# B&R Automation Studio project Lab1FuncBlocks
Automation Studio 4.5.2.102

## Configuration Config1

### Task classes (Cpu.sw)
```
Cyclic#4:
  Program <- Program.prg
Libraries: MotorCntrl
```

### Hardware
```
4PP065_0571_P74 : 4PP065.0571-P74 v1.1.2.0
  Simulation = 1
```

## Logical view

### Library Logical/Libraries/MotorCntrl (ANSIC)

#### MotorCntrl.fun - Exported functions and function blocks
```iecst
{REDUND_ERROR} {REDUND_UNREPLICABLE} FUNCTION_BLOCK FB_Motor (*Motor Model*) (*$GROUP=User,$CAT=User,$GROUPICON=User.png,$CATICON=User.png*)
	VAR_INPUT
		u : {REDUND_UNREPLICABLE} REAL; (*input voltage*)
	END_VAR
	VAR_OUTPUT
		w : {REDUND_UNREPLICABLE} REAL; (*rotation speed*)
		phi : {REDUND_UNREPLICABLE} REAL; (*position*)
	END_VAR
	VAR
		integrator : {REDUND_UNREPLICABLE} FB_Integrator; (*integrator*)
		Tm : {REDUND_UNREPLICABLE} REAL; (*Tm*)
		Ke : {REDUND_UNREPLICABLE} REAL; (*Ke*)
		dt : {REDUND_UNREPLICABLE} REAL; (*calc step*)
	END_VAR
END_FUNCTION_BLOCK

{REDUND_ERROR} {REDUND_UNREPLICABLE} FUNCTION_BLOCK FB_Integrator (*Integrator*) (*$GROUP=User,$CAT=User,$GROUPICON=User.png,$CATICON=User.png*)
	VAR_INPUT
		in : {REDUND_UNREPLICABLE} REAL; (*inp_integrator*)
	END_VAR
	VAR_OUTPUT
		out : {REDUND_UNREPLICABLE} REAL; (*out_integrator*)
	END_VAR
	VAR
		dt : {REDUND_UNREPLICABLE} REAL; (*calc_step*)
	END_VAR
END_FUNCTION_BLOCK

{REDUND_ERROR} FUNCTION_BLOCK FB_Regulator (*PI regulator*) (*$GROUP=User,$CAT=User,$GROUPICON=User.png,$CATICON=User.png*)
	VAR_INPUT
		e : {REDUND_UNREPLICABLE} REAL; (*Disagreement*)
	END_VAR
	VAR_OUTPUT
		u : {REDUND_UNREPLICABLE} REAL; (*voltage *)
	END_VAR
	VAR
		K_p : {REDUND_UNREPLICABLE} REAL; (*K_p*)
		K_i : {REDUND_UNREPLICABLE} REAL; (*K_i*)
		integrator : {REDUND_UNREPLICABLE} FB_Integrator; (*integrator*)
		iyOld : {REDUND_UNREPLICABLE} REAL; (*storing the value*)
		max_abs_value : {REDUND_UNREPLICABLE} REAL; (*edge of restriction block*)
		dt : {REDUND_UNREPLICABLE} REAL; (*calc_step*)
	END_VAR
END_FUNCTION_BLOCK
```

#### FB_Motor.c
```c
#include <bur/plctypes.h>
#ifdef __cplusplus
	extern "C"
	{
#endif
	#include "MotorCntrl.h"
#ifdef __cplusplus
	};
#endif
/* Motor Model */
void FB_Motor(struct FB_Motor* inst)
{
	inst->integrator.in = (inst->u / inst->Ke - inst->w) * inst->dt / inst->Tm;
	FB_Integrator(&(inst->integrator));
	inst->w = inst->integrator.out;
	inst->integrator.in = inst->w * inst->dt;
	FB_Integrator(&(inst->integrator));
	inst->phi = inst->integrator.out;
}
```

#### FB_Integrator.c
```c
#include <bur/plctypes.h>
#ifdef __cplusplus
	extern "C"
	{
#endif
	#include "MotorCntrl.h"
#ifdef __cplusplus
	};
#endif
/* Integrator */
void FB_Integrator(struct FB_Integrator* inst)
{
	inst->out +=  inst->in;
}
```

#### FB_Regulator.c
```c
#include <bur/plctypes.h>
#ifdef __cplusplus
	extern "C"
	{
#endif
	#include "MotorCntrl.h"
#ifdef __cplusplus
	};
#endif

void FB_Regulator(struct FB_Regulator* inst)
{

	REAL in_BON=0; REAL sum_after = 0;
	inst->integrator.in=inst->e * inst->K_i * inst->dt + inst->iyOld;
	FB_Integrator(&(inst->integrator));
	in_BON = inst-> e * inst->K_p;

	if(in_BON > inst->max_abs_value)
	{in_BON = inst->max_abs_value;}

	sum_after = in_BON + inst->integrator.out;
	if(sum_after > inst->max_abs_value)
	{inst->u = inst->max_abs_value;}
	else {inst->u = sum_after;}
	inst->iyOld =inst->u - sum_after;
}
```

### Program Logical/Program

#### Variables.var
```iecst
VAR
	speed : REAL;
	fb_motor_2 : FB_Motor;
	fb_motor : FB_Motor;
	fb_controller : FB_Regulator;
	enable : BOOL;
	count : INT;
END_VAR
```

#### Main.c
```c
#include <bur/plctypes.h>

#ifdef _DEFAULT_INCLUDES
	#include <AsDefault.h>
#endif

void _INIT ProgramInit(void)
{
	enable = 1;
	speed = 0;
	count = 0;

	fb_motor.u = 0;
	fb_motor.phi = 0;
	fb_motor.w = 0;
	fb_motor.Ke = 0.25;
	fb_motor.Tm = 0.1;
	fb_motor.dt = 0.02;;

	fb_motor_2.u = 0;
	fb_motor_2.phi = 0;
	fb_motor_2.w = 0;
	fb_motor_2.Ke = 0.25;
	fb_motor_2.Tm = 0.1;
	fb_motor_2.dt = 0.02;

	fb_controller.iyOld = 0;
	fb_controller.u = 0;
	/*fb_controller.K_p = fb_motor.Ke *fb_motor.Tm; */
	fb_controller.K_p = 0.025;
	/*fb_controller.K_i = fb_motor.Ke; */
	fb_controller.K_i = 0.25;
	fb_controller.max_abs_value=12;
	fb_controller.dt = 0.02;
}

void _CYCLIC ProgramCyclic(void)
{
	if(enable == 1)
	{
		/*
		count += 10;
		if(count<=5000)
		{
			speed=0;
		}
		else
		{
			speed=5;
			if(count >= 10000)
			{
				count = 0;
			}
		}
		*/

	/*need adjustment*/
		count += 100;
		if(count<5000)
		{
			speed=0;
		}
		else if( count >= 10000 && count <= 15000)
		{
			speed=5;
		}
		else {speed=0;}

		/*
		count += 100;
		if( (count >= 10000) && (count <=30000))
		{
			speed =3;
		}
		else {
			speed=0;
		}
		*/
		/* С регулятором: */
		fb_controller.e = speed - fb_motor.w;
		/*fb_controller.e = speed - fb_motor.phi;*/
		FB_Regulator(&fb_controller);
		fb_motor.u= fb_controller.u;
		FB_Motor(&fb_motor);

		/* Без регулятора: */
		fb_motor_2.u = speed - fb_motor_2.w;
		FB_Motor(&fb_motor_2);

	}

}

void _EXIT ProgramExit(void)
{

}
```

Listed in the project but not available here: Logical/Libraries/MotorCntrl/Types.typ, Logical/Libraries/MotorCntrl/Constants.var
